FUNCTION_BLOCK FB_FIFO_Lreal EXTENDS FB_Universal_FIFO IMPLEMENTS I_FIFO_Lreal
VAR_INPUT
  
END_VAR

VAR
  
END_VAR

VAR_OUTPUT
	OldestData : LREAL;
END_VAR
VAR PERSISTENT
	Queue : ARRAY[0..MaxQueueSize-1] OF LREAL;  // FIFO queue (size is 100 elements)
END_VAR



//    // Log new data only if LogData is TRUE
//    IF rTrigLogData.Q THEN
//        IF Count < MaxQueueSize THEN
//            Queue[Head] := NewEnergyData;
//            Head := (Head + 1) MOD MaxQueueSize;
//            Count := Count + 1;
//        ELSE
//            // FIFO is full, overwrite old data if needed
//            Tail := (Tail + 1) MOD MaxQueueSize;
//            Queue[Head] := NewEnergyData;
//            Head := (Head + 1) MOD MaxQueueSize;
//            // Tail position is updated
//        END_IF
//        DataReady := TRUE;  // New data is now ready to be processed
     
//    END_IF

    // Retrieve and manage oldest data for processing

// if dataready return true, else return false
METHOD  MR_AckGetValue : BOOL
VAR_INPUT
END_VAR
SUPER^.MR_AckGetValue();
  OldestData := Queue[Tail];
 MR_AckGetValue := true;
END_METHOD

METHOD MR_AddValue : BOOL
VAR_INPUT
		Value : LREAL;
END_VAR
  IF Count < MaxQueueSize THEN
            Queue[Head] := Value;
            Head := (Head + 1) MOD MaxQueueSize;
            Count := Count + 1;
  ELSE
            // FIFO is full, overwrite old data if needed
            Tail := (Tail + 1) MOD MaxQueueSize;
            Queue[Head] := Value;
            Head := (Head + 1) MOD MaxQueueSize;
            // Tail position is updated
			
  END_IF
  
  OldestData := Queue[Tail];
  bDataReady := TRUE; 
  
  
  MR_AddValue := true;
END_METHOD

// need overide to reset oldestValue
METHOD MR_Reset : BOOL
VAR_INPUT
END_VAR
SUPER^.MR_Reset();
OldestData := 0;
MR_Reset := true;
END_METHOD

PROPERTY oOldestValue : Lreal
GET
oOldestValue := OldestData;
END_GET
END_PROPERTY

END_FUNCTION_BLOCK

(* stored: Version 1.1.0.1, ProductVersion 3.1.4024.12
   POU FB_FIFO_Lreal: Id {8f3a32f0-7e00-4ebb-899d-be125261f986}, SpecialFunc None
   Method MR_AckGetValue: Id {09561704-badb-4272-b93c-ac7aae38809f}
   Method MR_AddValue: Id {ffe5f7f4-ae52-4ecc-8755-2ab6cb8cfce7}
   Method MR_Reset: Id {2a2b19b1-ebb1-4113-b1a5-5e202f98f473}
   Property oOldestValue: Id {98b612bb-2560-4227-bb88-040f3f05f6b2}
   Get Get: Id {4db1abac-4d66-4251-875f-070beb6efbbf} *)
